FUNCTION_BLOCK FB_OnSetpointCheck
VAR_INPUT
	fSP			: REAL; 
	fFB			: REAL;	
	fBand		: REAL;	
	tDelay		: TIME;	
END_VAR
VAR_OUTPUT
	bOnSP	: BOOL := FALSE;
	fCmd	: REAL;	
END_VAR 
VAR
	fbTon	: TON;
END_VAR

fCmd := fSP;

IF fFB > (fSP - fBand) AND fFB < (fSP + fBand) THEN
	fbTon(IN := TRUE, PT := tDelay);
ELSE
	fbTon(IN := FALSE);
END_IF

bOnSP := fbTon.Q;

END_FUNCTION_BLOCK

(* stored: Version 1.1.0.1, ProductVersion 3.1.4024.9
   POU FB_OnSetpointCheck: Id {4fe2bcd6-d66b-4da0-a242-ec88ace108d2}, SpecialFunc None *)
